TYPE E_StateAnalog : (
	eAnalog_Init,
	eAnalog_Start,
	eAnalog_LimitLow,
	eAnalog_LimitHigh,
	eAnalog_End
	);
END_TYPE

(* stored: Version 1.1.0.1, ProductVersion 3.1.4018.5
   DUT E_StateAnalog: Id {35c75778-9546-44a3-8d03-c2169abcf5e1} *)
